// TIA Portal V16 export
// export: Created 2024-12-03T15:41:40.1401816Z, ExportSetting WithDefaults, DisplayName Totally Integrated Automation Portal, DisplayVersion V16 Update 6, DisplayName TIA Portal Version Control Interface, DisplayVersion V16 Update 2, DisplayName TIA Portal Openness, DisplayVersion V16 Update 6, DisplayName TIA Portal Teamcenter Gateway, DisplayVersion V16, DisplayName SINAMICS Startdrive Advanced, DisplayVersion V16 Update 5, DisplayName SINAMICS Startdrive G130, G150, S120, S150, SINAMICS MV, S210, DisplayVersion V16 Update 5, DisplayName SINAMICS Startdrive G110M, G120, G120C, G120D, G120P, G115D, DisplayVersion V16 Update 5, DisplayName STEP 7 Professional, DisplayVersion V16 Update 6, DisplayName STEP 7 Safety, DisplayVersion V16, DisplayName WinCC Advanced / Unified PC, DisplayVersion V16 Update 6
FUNCTION_BLOCK "Settings_Convyors_Logic_FB"   // FB4, SCL
{ S7_Optimized_Access := 'TRUE' }
VERSION : 0.1
// stored: AutoNumber true, IsIECCheckEnabled false, IsRetainMemResEnabled false, MemoryReserve 100, SetENOAutomatically false, UDAEnableTagReadback false
   VAR
      settingsSaved : Bool;
   END_VAR
   VAR_TEMP
      T_SPEED : Real;
      T_mode : Int;
      T_RunIddle : Bool;
   END_VAR
BEGIN
   IF "HMI_DB".ReloadSettings.signal OR NOT #settingsSaved THEN

       REGION MODE

           #T_mode := "RUNTILLEND_MODE";

           "CONV_DB".CONV_101.Settings.Mode := #T_mode;

           #T_mode := "ZPA_TRAIN_MODE";

           "CONV_DB".CONV_102L.Settings.Mode := #T_mode;
           "CONV_DB".CONV_102R.Settings.Mode := #T_mode;
           "CONV_DB".CONV_103L.Settings.Mode := #T_mode;
           "CONV_DB".CONV_103R.Settings.Mode := #T_mode;
           "CONV_DB".CONV_104L.Settings.Mode := #T_mode;
           "CONV_DB".CONV_104R.Settings.Mode := #T_mode;
           "CONV_DB".CONV_105L.Settings.Mode := #T_mode;
           "CONV_DB".CONV_105R.Settings.Mode := #T_mode;
           "CONV_DB".CONV_106R.Settings.Mode := #T_mode;
           "CONV_DB".CONV_107R.Settings.Mode := #T_mode;
           "CONV_DB".CONV_108L.Settings.Mode := #T_mode;
           "CONV_DB".CONV_108R.Settings.Mode := #T_mode;
           "CONV_DB".CONV_109L.Settings.Mode := #T_mode;
           "CONV_DB".CONV_109R.Settings.Mode := #T_mode;
           "CONV_DB".CONV_110L.Settings.Mode := #T_mode;
           "CONV_DB".CONV_110R.Settings.Mode := #T_mode;
           "CONV_DB".CONV_111L.Settings.Mode := #T_mode;
           "CONV_DB".CONV_111R.Settings.Mode := #T_mode;
           "CONV_DB".CONV_112R.Settings.Mode := #T_mode;
           "CONV_DB".CONV_113L.Settings.Mode := #T_mode;
           "CONV_DB".CONV_113R.Settings.Mode := #T_mode;
           "CONV_DB".CONV_114L.Settings.Mode := #T_mode;
           "CONV_DB".CONV_114R.Settings.Mode := #T_mode;
           "CONV_DB".CONV_115L.Settings.Mode := #T_mode;
           "CONV_DB".CONV_115R.Settings.Mode := #T_mode;
           "CONV_DB".CONV_201R_BELTS.Settings.Mode := #T_mode;
           "CONV_DB".CONV_203R_BELTS.Settings.Mode := #T_mode;
           "CONV_DB".CONV_301R.Settings.Mode := #T_mode;
           "CONV_DB".CONV_302L.Settings.Mode := #T_mode;
           "CONV_DB".CONV_302R.Settings.Mode := #T_mode;
           "CONV_DB".CONV_303L.Settings.Mode := #T_mode;
           "CONV_DB".CONV_303R.Settings.Mode := #T_mode;
           "CONV_DB".CONV_304L.Settings.Mode := #T_mode;
           "CONV_DB".CONV_304R.Settings.Mode := #T_mode;
           "CONV_DB".CONV_305R.Settings.Mode := #T_mode;

       END_REGION

       REGION SPEED

           #T_SPEED := #T_SPEED;

           "CONV_DB".CONV_101.Settings.Speed.speed := #T_SPEED;
           "CONV_DB".CONV_102L.Settings.Speed.speed := #T_SPEED;
           "CONV_DB".CONV_102R.Settings.Speed.speed := #T_SPEED;
           "CONV_DB".CONV_103L.Settings.Speed.speed := #T_SPEED;
           "CONV_DB".CONV_103R.Settings.Speed.speed := #T_SPEED;
           "CONV_DB".CONV_104L.Settings.Speed.speed := #T_SPEED;
           "CONV_DB".CONV_104R.Settings.Speed.speed := #T_SPEED;
           "CONV_DB".CONV_105L.Settings.Speed.speed := #T_SPEED;
           "CONV_DB".CONV_105R.Settings.Speed.speed := #T_SPEED;
           "CONV_DB".CONV_106R.Settings.Speed.speed := #T_SPEED;
           "CONV_DB".CONV_107R.Settings.Speed.speed := #T_SPEED;
           "CONV_DB".CONV_108L.Settings.Speed.speed := #T_SPEED;
           "CONV_DB".CONV_108R.Settings.Speed.speed := #T_SPEED;
           "CONV_DB".CONV_109L.Settings.Speed.speed := #T_SPEED;
           "CONV_DB".CONV_109R.Settings.Speed.speed := #T_SPEED;
           "CONV_DB".CONV_110L.Settings.Speed.speed := #T_SPEED;
           "CONV_DB".CONV_110R.Settings.Speed.speed := #T_SPEED;
           "CONV_DB".CONV_111L.Settings.Speed.speed := #T_SPEED;
           "CONV_DB".CONV_111R.Settings.Speed.speed := #T_SPEED;
           "CONV_DB".CONV_112R.Settings.Speed.speed := #T_SPEED;
           "CONV_DB".CONV_113L.Settings.Speed.speed := #T_SPEED;
           "CONV_DB".CONV_113R.Settings.Speed.speed := #T_SPEED;
           "CONV_DB".CONV_114L.Settings.Speed.speed := #T_SPEED;
           "CONV_DB".CONV_114R.Settings.Speed.speed := #T_SPEED;
           "CONV_DB".CONV_115L.Settings.Speed.speed := #T_SPEED;
           "CONV_DB".CONV_115R.Settings.Speed.speed := #T_SPEED;
           "CONV_DB".CONV_201R_BELTS.Settings.Speed.speed := #T_SPEED;
           "CONV_DB".CONV_203R_BELTS.Settings.Speed.speed := #T_SPEED;
           "CONV_DB".CONV_301R.Settings.Speed.speed := #T_SPEED;
           "CONV_DB".CONV_302L.Settings.Speed.speed := #T_SPEED;
           "CONV_DB".CONV_302R.Settings.Speed.speed := #T_SPEED;
           "CONV_DB".CONV_303L.Settings.Speed.speed := #T_SPEED;
           "CONV_DB".CONV_303R.Settings.Speed.speed := #T_SPEED;
           "CONV_DB".CONV_304L.Settings.Speed.speed := #T_SPEED;
           "CONV_DB".CONV_304R.Settings.Speed.speed := #T_SPEED;
           "CONV_DB".CONV_305R.Settings.Speed.speed := #T_SPEED;


       END_REGION

       REGION RUN IDDLE

           #T_RunIddle := 1;

           "CONV_DB".CONV_101.Settings.RunIddle := #T_RunIddle;
           "CONV_DB".CONV_102L.Settings.RunIddle := #T_RunIddle;
           "CONV_DB".CONV_102R.Settings.RunIddle := #T_RunIddle;
           "CONV_DB".CONV_103L.Settings.RunIddle := #T_RunIddle;
           "CONV_DB".CONV_103R.Settings.RunIddle := #T_RunIddle;
           "CONV_DB".CONV_104L.Settings.RunIddle := #T_RunIddle;
           "CONV_DB".CONV_104R.Settings.RunIddle := #T_RunIddle;
           "CONV_DB".CONV_105L.Settings.RunIddle := #T_RunIddle;
           "CONV_DB".CONV_105R.Settings.RunIddle := #T_RunIddle;
           "CONV_DB".CONV_106R.Settings.RunIddle := #T_RunIddle;
           "CONV_DB".CONV_107R.Settings.RunIddle := #T_RunIddle;
           "CONV_DB".CONV_108L.Settings.RunIddle := #T_RunIddle;
           "CONV_DB".CONV_108R.Settings.RunIddle := #T_RunIddle;
           "CONV_DB".CONV_109L.Settings.RunIddle := #T_RunIddle;
           "CONV_DB".CONV_109R.Settings.RunIddle := #T_RunIddle;
           "CONV_DB".CONV_110L.Settings.RunIddle := #T_RunIddle;
           "CONV_DB".CONV_110R.Settings.RunIddle := #T_RunIddle;
           "CONV_DB".CONV_111L.Settings.RunIddle := #T_RunIddle;
           "CONV_DB".CONV_111R.Settings.RunIddle := #T_RunIddle;
           "CONV_DB".CONV_112R.Settings.RunIddle := #T_RunIddle;
           "CONV_DB".CONV_113L.Settings.RunIddle := #T_RunIddle;
           "CONV_DB".CONV_113R.Settings.RunIddle := #T_RunIddle;
           "CONV_DB".CONV_114L.Settings.RunIddle := #T_RunIddle;
           "CONV_DB".CONV_114R.Settings.RunIddle := #T_RunIddle;
           "CONV_DB".CONV_115L.Settings.RunIddle := #T_RunIddle;
           "CONV_DB".CONV_115R.Settings.RunIddle := #T_RunIddle;
           "CONV_DB".CONV_201R_BELTS.Settings.RunIddle := #T_RunIddle;
           "CONV_DB".CONV_203R_BELTS.Settings.RunIddle := #T_RunIddle;
           "CONV_DB".CONV_301R.Settings.RunIddle := #T_RunIddle;
           "CONV_DB".CONV_302L.Settings.RunIddle := #T_RunIddle;
           "CONV_DB".CONV_302R.Settings.RunIddle := #T_RunIddle;
           "CONV_DB".CONV_303L.Settings.RunIddle := #T_RunIddle;
           "CONV_DB".CONV_303R.Settings.RunIddle := #T_RunIddle;
           "CONV_DB".CONV_304L.Settings.RunIddle := #T_RunIddle;
           "CONV_DB".CONV_304R.Settings.RunIddle := #T_RunIddle;
           "CONV_DB".CONV_305R.Settings.RunIddle := #T_RunIddle;

       END_REGION

   END_IF;
END_FUNCTION_BLOCK
